(* Logix 5000 project; controller AdvManLab vendor 1 type 14 code 158 rev 28.12; software revision 28.01; part 7 of 13 *)
(* tags used below, declared in another part *)
   R6Z_Current_Part_NO : SINT;
   R6Z_Current_Process_NO : SINT;
   R6Z_Process : BOOL;
   R6Z_Read : BOOL;
   R6Z_Read_Finished : BOOL;
   R6Z_Write_Pass : BOOL;
   ABBLoopVFD : PF525_Faceplate_AOI;
   BobsBits : DINT;
   C21PartInTransit : TIMER;
   C23PartInTransit : TIMER;
   C2HoldBack : PalletStop;
   C2RobotStop : PalletStop;
   C2RobotStopPalletTransit : TIMER;
   C2RobotStopRetractConditions : BOOL;
   C31DiverterHoldBack : PalletStop;
   C31PartInTransit : TIMER;
   Cell_2 : Fanuc_Cell;
   Cloud_R1Z_TagPresent : BOOL;
   Cloud_R1Z_Timer : TIMER;
   Cloud_R2Z_TagPresent : BOOL;
   Cloud_R2Z_Timer : TIMER;
   Cloud_R3Z_TagPresent : BOOL;
   Cloud_R3Z_Timer : TIMER;
   Cloud_R4Z_TagPresent : BOOL;
   Cloud_R4Z_Timer : TIMER;
   Cloud_R5Z_TagPresent : BOOL;
   Cloud_R5Z_Timer : TIMER;
   Cloud_R6Z_TagPresent : BOOL;
   Cloud_R6Z_Timer : TIMER;
   CNC1Bools : DINT;
   CNC2Bools : DINT;
   CNC3Bools : DINT;
   CNC_1_ProgToRun : DINT;
   CNC_2_ProgToRun : DINT;   // G-Code Program Number for CNC to run TO CNC
   CNC_3_Done : BOOL;   // CNC 3 has completed cutting the part
   CNC_3_ProgToRun : DINT;   // G-code program number to be paassed to CNC to run
   CNC_4_Done : BOOL;   // CNC 4 has completed cutting the part
   Comm_Fault_Sts_Timer2 : TIMER;
   Comm_Status : DINT;
   Comm_Status2 : DINT;
   DeBounce3 : TIMER;
   DeBounce4 : TIMER;
   Fault_Code2 : DINT;
   FaultReset : BOOL;
   FltMsg2 : MESSAGE;
   FromCNC1 : CNC_Datablock;   // Data From CNC1
   FromCNC2 : CNC_Datablock;   // Data From CNC2
   FromCNC3 : CNC_Datablock;   // Data From CNC3
   FromCNC4 : CNC_Datablock;   // Data From CNC4
   HMI_Mode : DINT;
   Mode_Auto : BOOL;
   Mode_Semi : BOOL;
   Mode_Start : BOOL;
   ONS : DINT;
   PF525_AlarmName2 : STRING;
   PowerFlexAlarmName2 : STRING;
   PowerFlexAlarmTrigger2 : DINT;
   PPX2 : ALIAS FOR Conv_N053:3:I.0;   // Sensor Pallet Stop RFID2 (Cell 2 Hold Back Stop)
   PPX3 : ALIAS FOR Conv_N053:3:I.1;   // Sensor Pallet Stop RFID3 (Cell 2 Fanuc Robot Stop)
   R2Z_Read_Finished : BOOL;
   R3J_Current_Part_NO : SINT;
   R3J_Current_Process_NO : SINT;
   R3J_Read_Finished : BOOL;
   R3J_Write_Pass : BOOL;
   RelC2HoldBack : TIMER;
   RFIDTP1 : ALIAS FOR RFID_N054:I.Channel[0].TagPresent;   // RFID Tag at Cell 1 Stop
   RFIDTP2 : ALIAS FOR RFID_N054:I.Channel[1].TagPresent;   // RFID Tag at Cell 2 Hold Back Stop
   RFIDTP3 : ALIAS FOR RFID_N055:I.Channel[0].TagPresent;   // RFID Tag at Cell 2 Stop
   RFIDTP4 : ALIAS FOR RFID_N055:I.Channel[1].TagPresent;   // RFID Tag at Cell C23 Hold Back Stop
   RFIDTP5 : ALIAS FOR RFID_N056:I.Channel[0].TagPresent;   // RFID Tag at Cell 3 Stop
   RFIDTP6 : ALIAS FOR RFID_N056:I.Channel[1].TagPresent;
   Robot1_Busy_ZZ : BOOL;
   Robot2_Busy_ZZ : BOOL;
   RunPartOnCNC1 : BOOL;
   RunPartOnCNC2 : BOOL;
   RunpartOnCNC3 : BOOL;
   RunPartOnCNC4 : BOOL;
   ToCNC1 : CNC_Datablock;   // Data To CNC1
   ToCNC2 : CNC_Datablock;   // Data To CNC2
   ToCNC3 : CNC_Datablock;   // Data To CNC3
(* MainProgram, continued *)

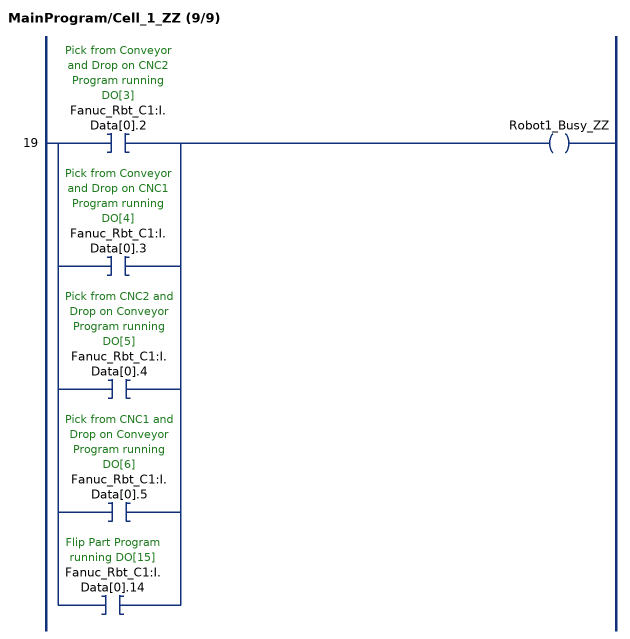
   [picture p119: MainProgram/Cell_1_ZZ rungs 19-19]
   19: [XIC(Fanuc_Rbt_C1:I.Data[0].2) ,XIC(Fanuc_Rbt_C1:I.Data[0].3) ,XIC(Fanuc_Rbt_C1:I.Data[0].4) ,XIC(Fanuc_Rbt_C1:I.Data[0].5) ,XIC(Fanuc_Rbt_C1:I.Data[0].14) ]OTE(Robot1_Busy_ZZ);
END_ROUTINE

ROUTINE Cell_2_ZZ   (* ladder *)
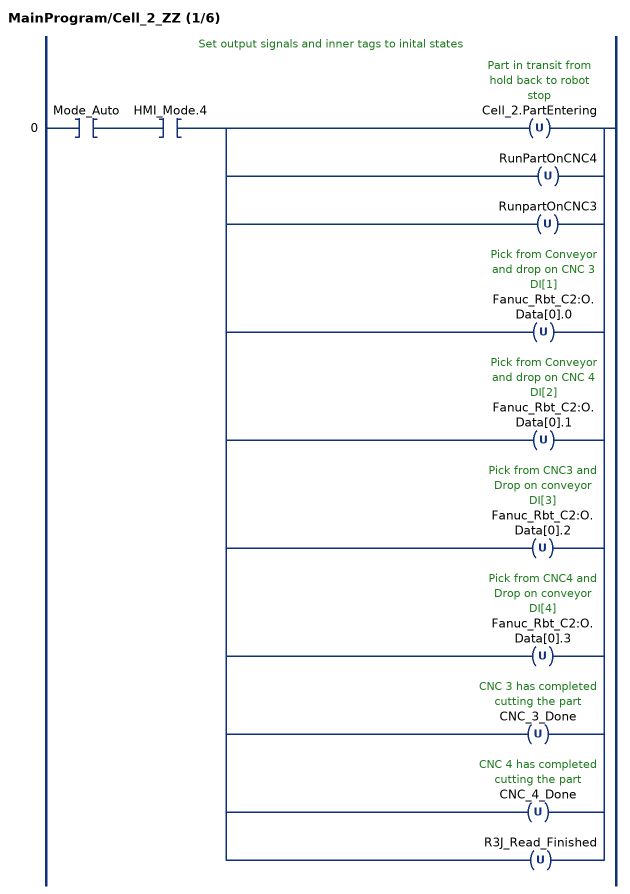
   // Set output signals and inner tags to inital states
   0: XIC(Mode_Auto)XIC(HMI_Mode.4)[OTU(Cell_2.PartEntering) ,OTU(RunPartOnCNC4) ,OTU(RunpartOnCNC3) ,OTU(Fanuc_Rbt_C2:O.Data[0].0) ,OTU(Fanuc_Rbt_C2:O.Data[0].1) ,OTU(Fanuc_Rbt_C2:O.Data[0].2) ,OTU(Fanuc_Rbt_C2:O.Data[0].3) ,OTU(CNC_3_Done) ,OTU(CNC_4_Done) ,OTU(R3J_Read_Finished) ];
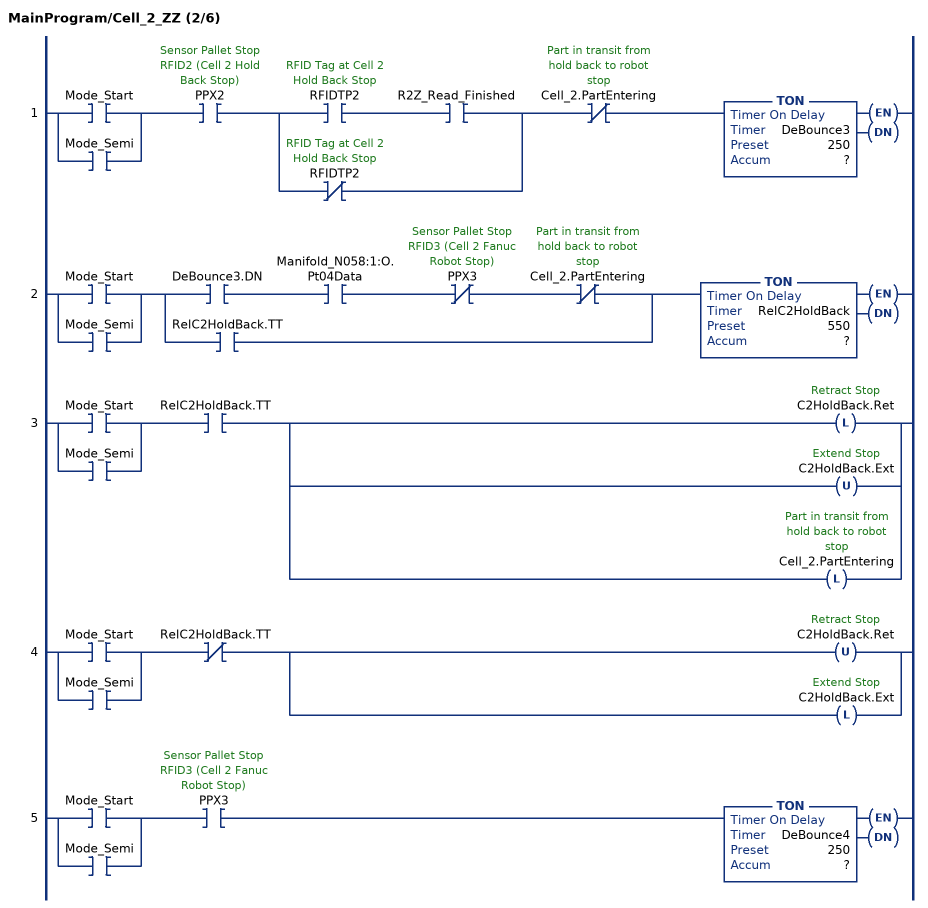
   1: [XIC(Mode_Start) ,XIC(Mode_Semi) ]XIC(PPX2)[XIC(RFIDTP2) XIC(R2Z_Read_Finished) ,XIO(RFIDTP2) ]XIO(Cell_2.PartEntering)TON(DeBounce3,?,?);
   2: [XIC(Mode_Start) ,XIC(Mode_Semi) ][XIC(DeBounce3.DN) XIC(Manifold_N058:1:O.Pt04Data) XIO(PPX3) XIO(Cell_2.PartEntering) ,XIC(RelC2HoldBack.TT) ]TON(RelC2HoldBack,?,?);
   3: [XIC(Mode_Start) ,XIC(Mode_Semi) ]XIC(RelC2HoldBack.TT)[OTL(C2HoldBack.Ret) ,OTU(C2HoldBack.Ext) ,OTL(Cell_2.PartEntering) ];
   4: [XIC(Mode_Start) ,XIC(Mode_Semi) ]XIO(RelC2HoldBack.TT)[OTU(C2HoldBack.Ret) ,OTL(C2HoldBack.Ext) ];
   5: [XIC(Mode_Start) ,XIC(Mode_Semi) ]XIC(PPX3)TON(DeBounce4,?,?);
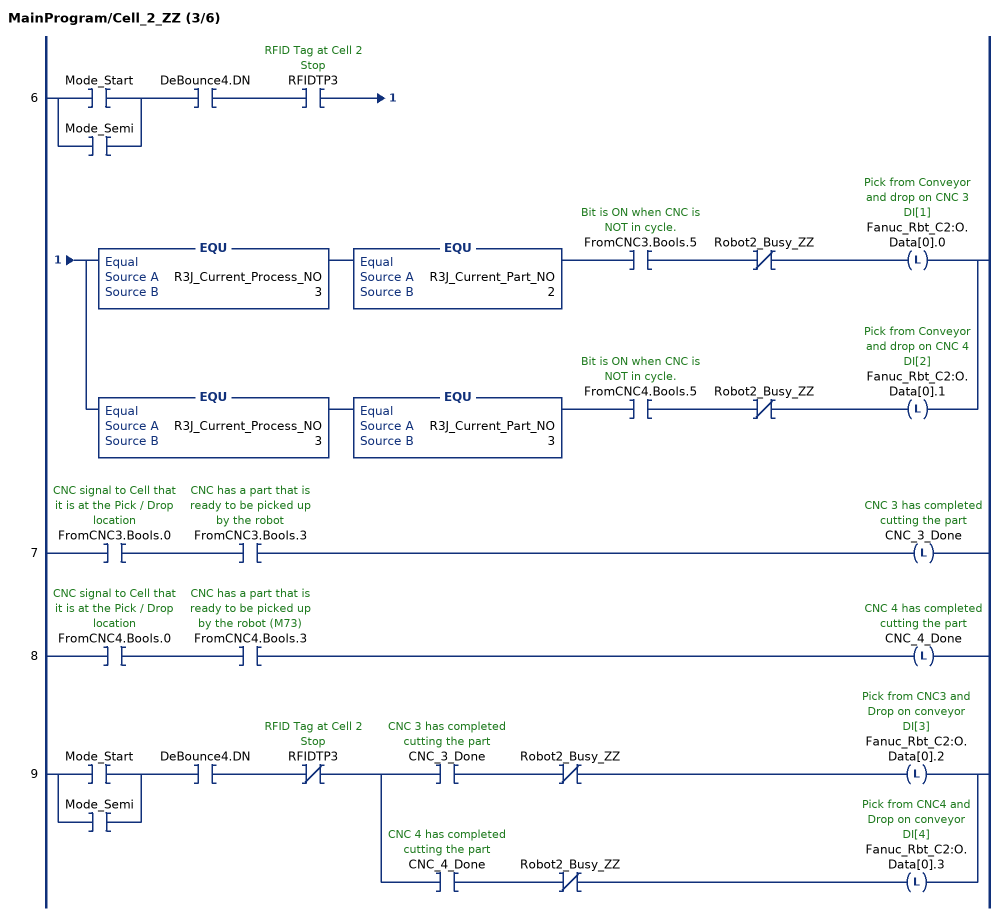
   6: [XIC(Mode_Start) ,XIC(Mode_Semi) ]XIC(DeBounce4.DN)XIC(RFIDTP3)[EQU(R3J_Current_Process_NO,3) EQU(R3J_Current_Part_NO,2) XIC(FromCNC3.Bools.5) XIO(Robot2_Busy_ZZ) OTL(Fanuc_Rbt_C2:O.Data[0].0) ,EQU(R3J_Current_Process_NO,3) EQU(R3J_Current_Part_NO,3) XIC(FromCNC4.Bools.5) XIO(Robot2_Busy_ZZ) OTL(Fanuc_Rbt_C2:O.Data[0].1) ];
   7: XIC(FromCNC3.Bools.0)XIC(FromCNC3.Bools.3)OTL(CNC_3_Done);
   8: XIC(FromCNC4.Bools.0)XIC(FromCNC4.Bools.3)OTL(CNC_4_Done);
   9: [XIC(Mode_Start) ,XIC(Mode_Semi) ]XIC(DeBounce4.DN)XIO(RFIDTP3)[XIC(CNC_3_Done) XIO(Robot2_Busy_ZZ) OTL(Fanuc_Rbt_C2:O.Data[0].2) ,XIC(CNC_4_Done) XIO(Robot2_Busy_ZZ) OTL(Fanuc_Rbt_C2:O.Data[0].3) ];
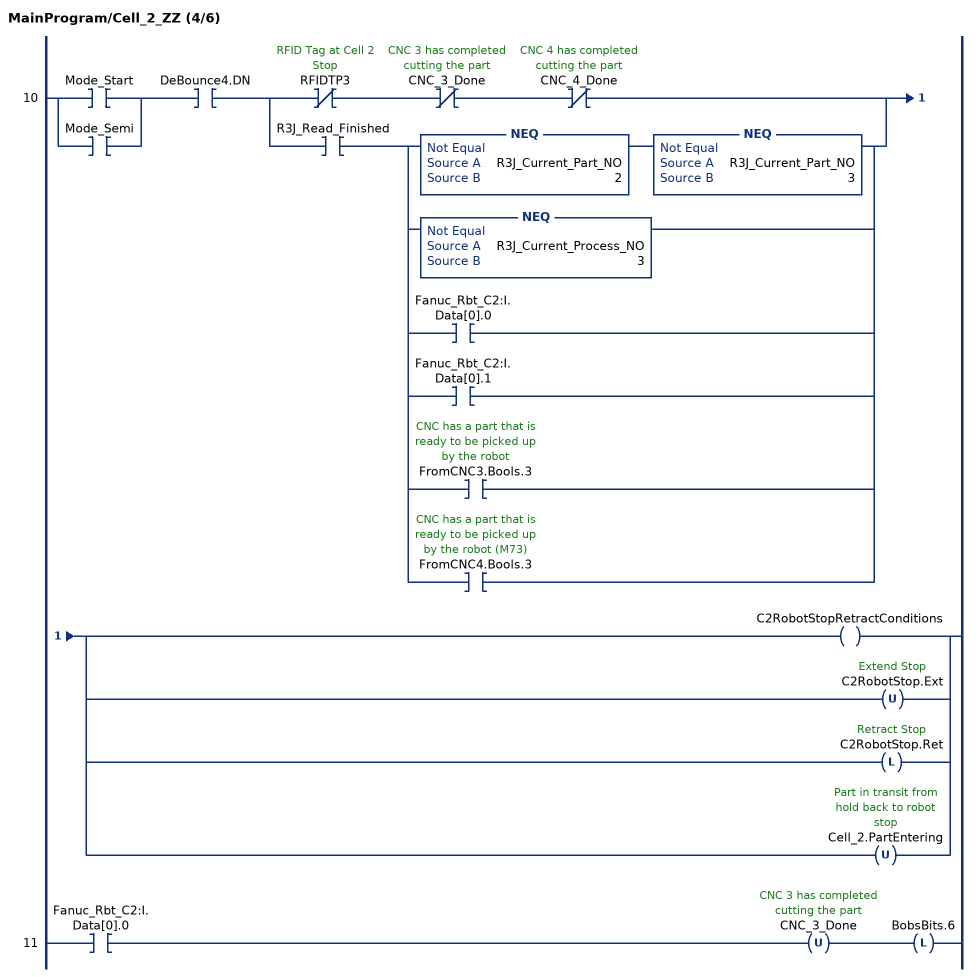
   10: [XIC(Mode_Start) ,XIC(Mode_Semi) ]XIC(DeBounce4.DN)[XIO(RFIDTP3) XIO(CNC_3_Done) XIO(CNC_4_Done) ,XIC(R3J_Read_Finished) [NEQ(R3J_Current_Part_NO,2) NEQ(R3J_Current_Part_NO,3) ,NEQ(R3J_Current_Process_NO,3) ,XIC(Fanuc_Rbt_C2:I.Data[0].0) ,XIC(Fanuc_Rbt_C2:I.Data[0].1) ,[XIC(FromCNC3.Bools.3) ,XIC(FromCNC4.Bools.3) ] ] ][OTE(C2RobotStopRetractConditions) ,OTU(C2RobotStop.Ext) ,OTL(C2RobotStop.Ret) ,OTU(Cell_2.PartEntering) ];
   11: XIC(Fanuc_Rbt_C2:I.Data[0].0)OTU(CNC_3_Done)OTL(BobsBits.6);
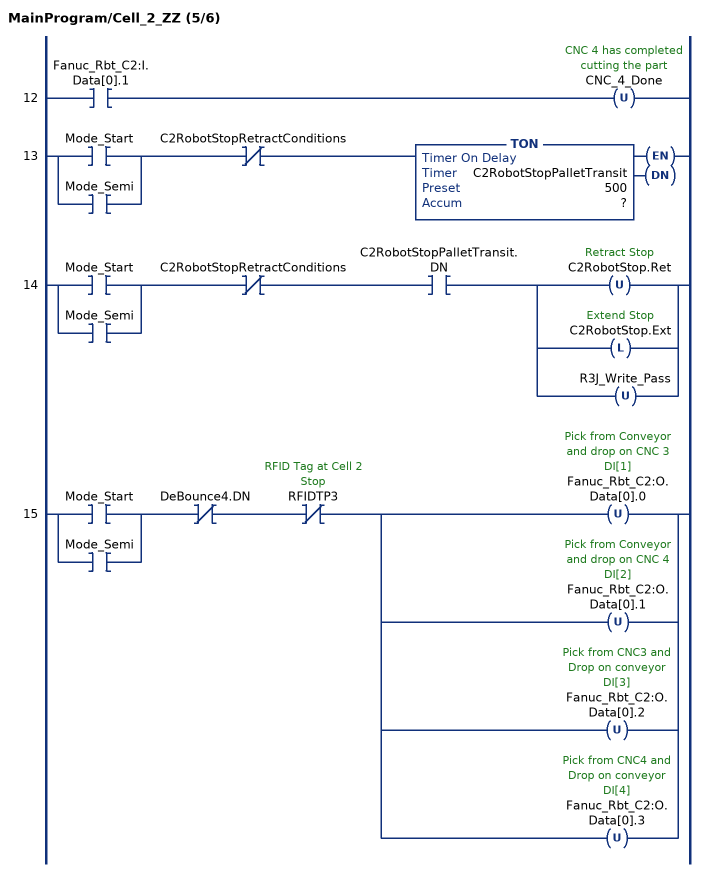
   12: XIC(Fanuc_Rbt_C2:I.Data[0].1)OTU(CNC_4_Done);
   13: [XIC(Mode_Start) ,XIC(Mode_Semi) ]XIO(C2RobotStopRetractConditions)TON(C2RobotStopPalletTransit,?,?);
   14: [XIC(Mode_Start) ,XIC(Mode_Semi) ]XIO(C2RobotStopRetractConditions)XIC(C2RobotStopPalletTransit.DN)[OTU(C2RobotStop.Ret) ,OTL(C2RobotStop.Ext) ,OTU(R3J_Write_Pass) ];
   15: [XIC(Mode_Start) ,XIC(Mode_Semi) ]XIO(DeBounce4.DN)XIO(RFIDTP3)[OTU(Fanuc_Rbt_C2:O.Data[0].0) ,OTU(Fanuc_Rbt_C2:O.Data[0].1) ,OTU(Fanuc_Rbt_C2:O.Data[0].2) ,OTU(Fanuc_Rbt_C2:O.Data[0].3) ];
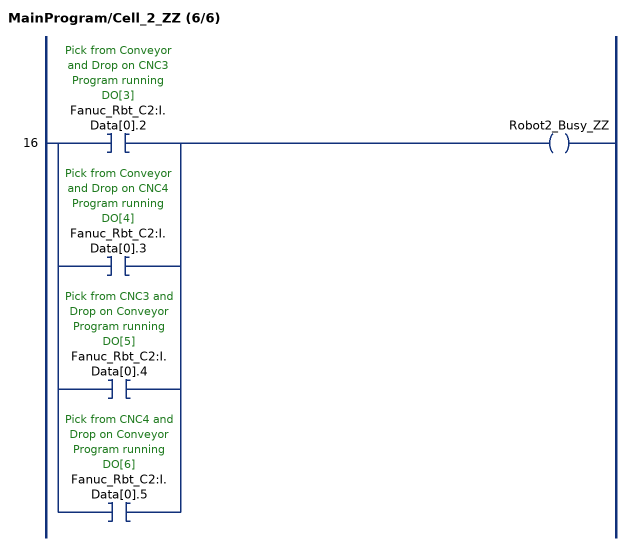
   16: [XIC(Fanuc_Rbt_C2:I.Data[0].2) ,XIC(Fanuc_Rbt_C2:I.Data[0].3) ,XIC(Fanuc_Rbt_C2:I.Data[0].4) ,XIC(Fanuc_Rbt_C2:I.Data[0].5) ]OTE(Robot2_Busy_ZZ);
END_ROUTINE

ROUTINE Cell_3_VFD   (* ladder *)
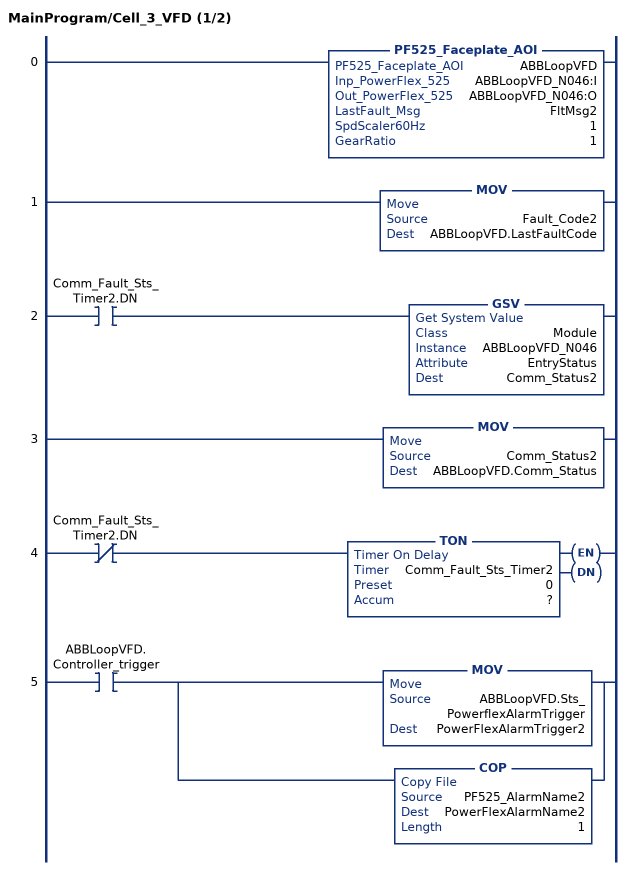
   0: PF525_Faceplate_AOI(ABBLoopVFD,ABBLoopVFD_N046:I,ABBLoopVFD_N046:O,FltMsg2,1,1);
   1: MOV(Fault_Code2,ABBLoopVFD.LastFaultCode);
   2: XIC(Comm_Fault_Sts_Timer2.DN)GSV(Module,ABBLoopVFD_N046,EntryStatus,Comm_Status2);
   3: MOV(Comm_Status2,ABBLoopVFD.Comm_Status);
   4: XIO(Comm_Fault_Sts_Timer2.DN)TON(Comm_Fault_Sts_Timer2,?,?);
   5: XIC(ABBLoopVFD.Controller_trigger)[MOV(ABBLoopVFD.Sts_PowerflexAlarmTrigger,PowerFlexAlarmTrigger2) ,COP(PF525_AlarmName2,PowerFlexAlarmName2,1) ];
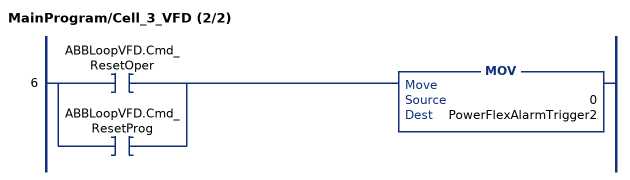
   6: [XIC(ABBLoopVFD.Cmd_ResetOper) ,XIC(ABBLoopVFD.Cmd_ResetProg) ]MOV(0,PowerFlexAlarmTrigger2);
END_ROUTINE

ROUTINE Cell_3_ZZ   (* ladder *)
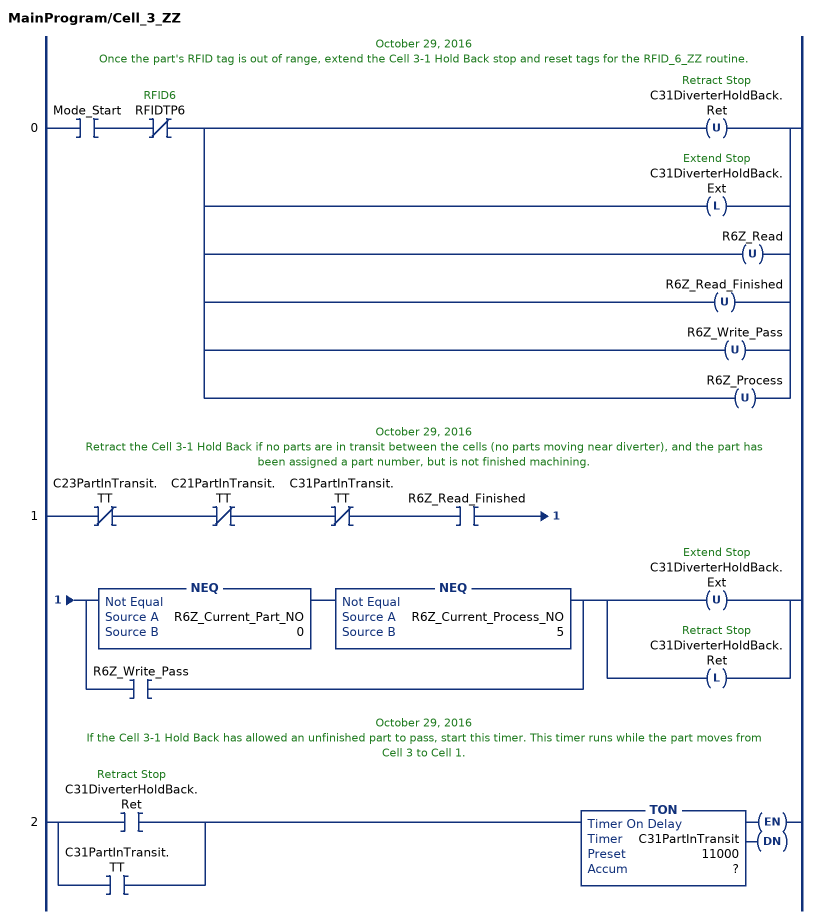
   // October 29, 2016
   // Once the part's RFID tag is out of range, extend the Cell 3-1 Hold Back stop and reset tags for the RFID_6_ZZ routine.
   0: XIC(Mode_Start)XIO(RFIDTP6)[OTU(C31DiverterHoldBack.Ret) ,OTL(C31DiverterHoldBack.Ext) ,OTU(R6Z_Read) ,OTU(R6Z_Read_Finished) ,OTU(R6Z_Write_Pass) ,OTU(R6Z_Process) ];
   // October 29, 2016
   // Retract the Cell 3-1 Hold Back if no parts are in transit between the cells (no parts moving near diverter), and the part has been assigned a part number, but is not finished machining.
   1: XIO(C23PartInTransit.TT)XIO(C21PartInTransit.TT)XIO(C31PartInTransit.TT)XIC(R6Z_Read_Finished)[NEQ(R6Z_Current_Part_NO,0) NEQ(R6Z_Current_Process_NO,5) ,XIC(R6Z_Write_Pass) ][OTU(C31DiverterHoldBack.Ext) ,OTL(C31DiverterHoldBack.Ret) ];
   // October 29, 2016
   // If the Cell 3-1 Hold Back has allowed an unfinished part to pass, start this timer. This timer runs while the part moves from Cell 3 to Cell 1.
   2: [XIC(C31DiverterHoldBack.Ret) ,XIC(C31PartInTransit.TT) ]TON(C31PartInTransit,?,?);
END_ROUTINE

ROUTINE Cloud_Team_ZZ   (* ladder *)
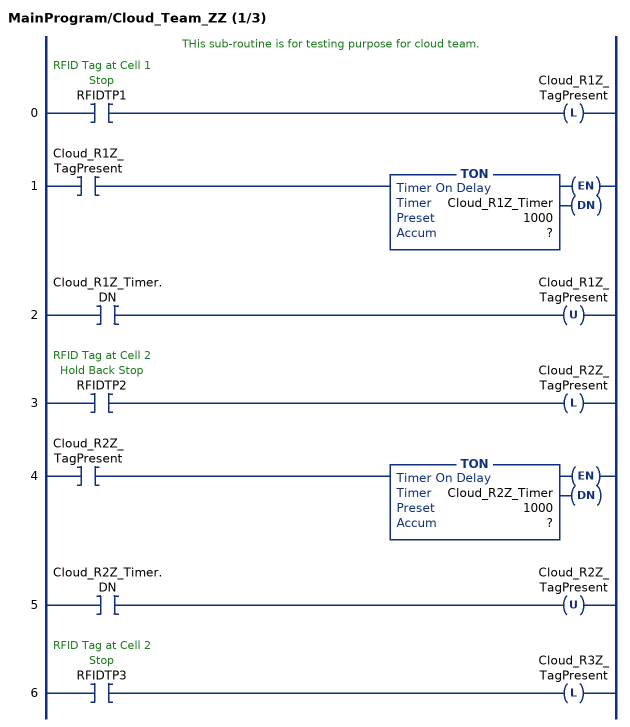
   // THis sub-routine is for testing purpose for cloud team.
   0: XIC(RFIDTP1)OTL(Cloud_R1Z_TagPresent);
   1: XIC(Cloud_R1Z_TagPresent)TON(Cloud_R1Z_Timer,?,?);
   2: XIC(Cloud_R1Z_Timer.DN)OTU(Cloud_R1Z_TagPresent);
   3: XIC(RFIDTP2)OTL(Cloud_R2Z_TagPresent);
   4: XIC(Cloud_R2Z_TagPresent)TON(Cloud_R2Z_Timer,?,?);
   5: XIC(Cloud_R2Z_Timer.DN)OTU(Cloud_R2Z_TagPresent);
   6: XIC(RFIDTP3)OTL(Cloud_R3Z_TagPresent);
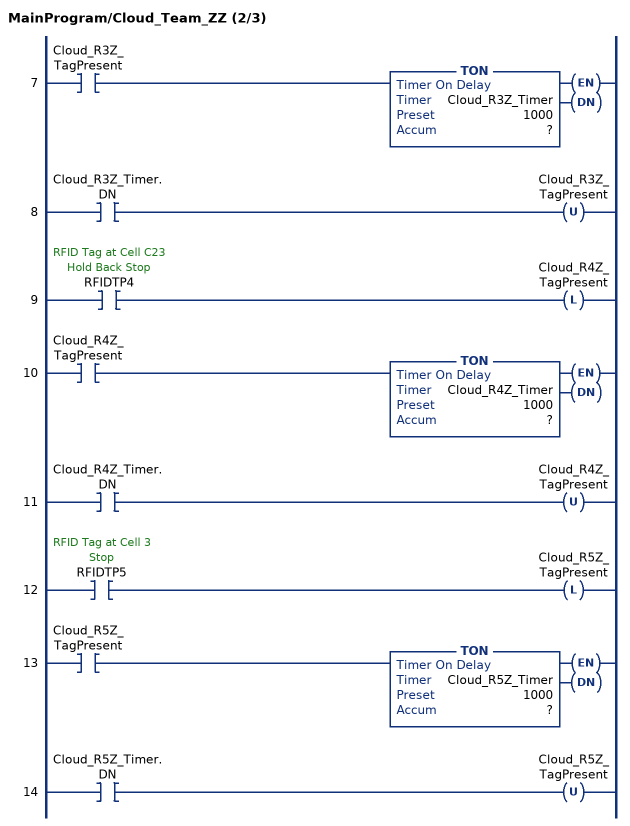
   7: XIC(Cloud_R3Z_TagPresent)TON(Cloud_R3Z_Timer,?,?);
   8: XIC(Cloud_R3Z_Timer.DN)OTU(Cloud_R3Z_TagPresent);
   9: XIC(RFIDTP4)OTL(Cloud_R4Z_TagPresent);
   10: XIC(Cloud_R4Z_TagPresent)TON(Cloud_R4Z_Timer,?,?);
   11: XIC(Cloud_R4Z_Timer.DN)OTU(Cloud_R4Z_TagPresent);
   12: XIC(RFIDTP5)OTL(Cloud_R5Z_TagPresent);
   13: XIC(Cloud_R5Z_TagPresent)TON(Cloud_R5Z_Timer,?,?);
   14: XIC(Cloud_R5Z_Timer.DN)OTU(Cloud_R5Z_TagPresent);
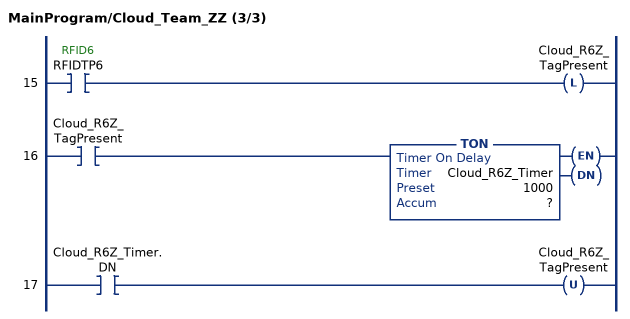
   15: XIC(RFIDTP6)OTL(Cloud_R6Z_TagPresent);
   16: XIC(Cloud_R6Z_TagPresent)TON(Cloud_R6Z_Timer,?,?);
   17: XIC(Cloud_R6Z_Timer.DN)OTU(Cloud_R6Z_TagPresent);
END_ROUTINE

ROUTINE CNC1   (* ladder *)
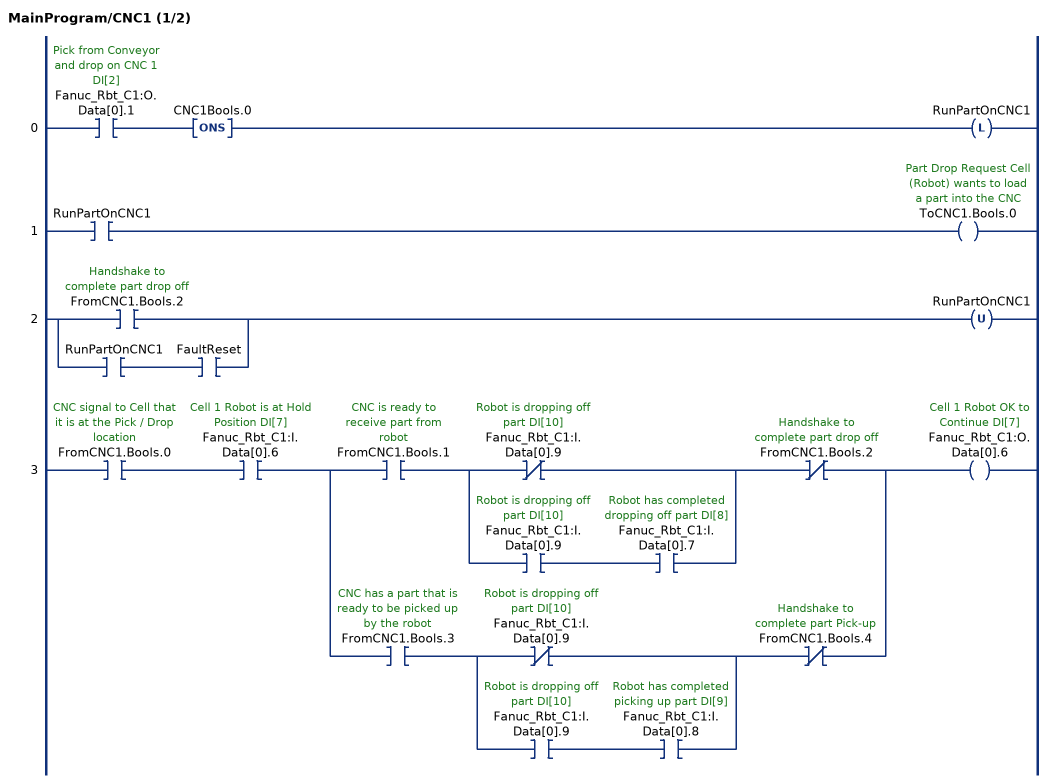
   0: XIC(Fanuc_Rbt_C1:O.Data[0].1)ONS(CNC1Bools.0)OTL(RunPartOnCNC1);
   1: XIC(RunPartOnCNC1)OTE(ToCNC1.Bools.0);
   2: [XIC(FromCNC1.Bools.2) ,XIC(RunPartOnCNC1) XIC(FaultReset) ]OTU(RunPartOnCNC1);
   3: XIC(FromCNC1.Bools.0)XIC(Fanuc_Rbt_C1:I.Data[0].6)[XIC(FromCNC1.Bools.1) [XIO(Fanuc_Rbt_C1:I.Data[0].9) ,XIC(Fanuc_Rbt_C1:I.Data[0].9) XIC(Fanuc_Rbt_C1:I.Data[0].7) ] XIO(FromCNC1.Bools.2) ,XIC(FromCNC1.Bools.3) [XIO(Fanuc_Rbt_C1:I.Data[0].9) ,XIC(Fanuc_Rbt_C1:I.Data[0].9) XIC(Fanuc_Rbt_C1:I.Data[0].8) ] XIO(FromCNC1.Bools.4) ]OTE(Fanuc_Rbt_C1:O.Data[0].6);
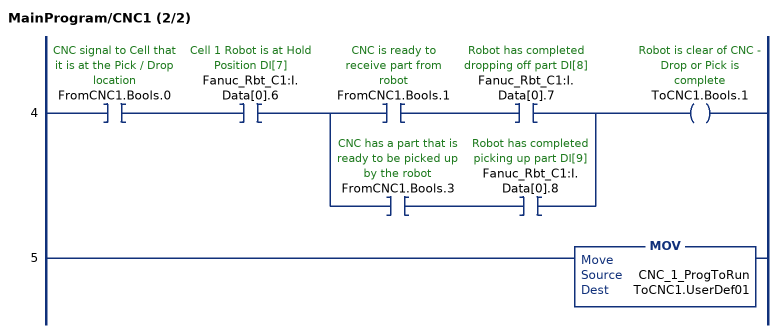
   4: XIC(FromCNC1.Bools.0)XIC(Fanuc_Rbt_C1:I.Data[0].6)[XIC(FromCNC1.Bools.1) XIC(Fanuc_Rbt_C1:I.Data[0].7) ,XIC(FromCNC1.Bools.3) XIC(Fanuc_Rbt_C1:I.Data[0].8) ]OTE(ToCNC1.Bools.1);
   5: MOV(CNC_1_ProgToRun,ToCNC1.UserDef01);
END_ROUTINE

ROUTINE CNC2   (* ladder *)
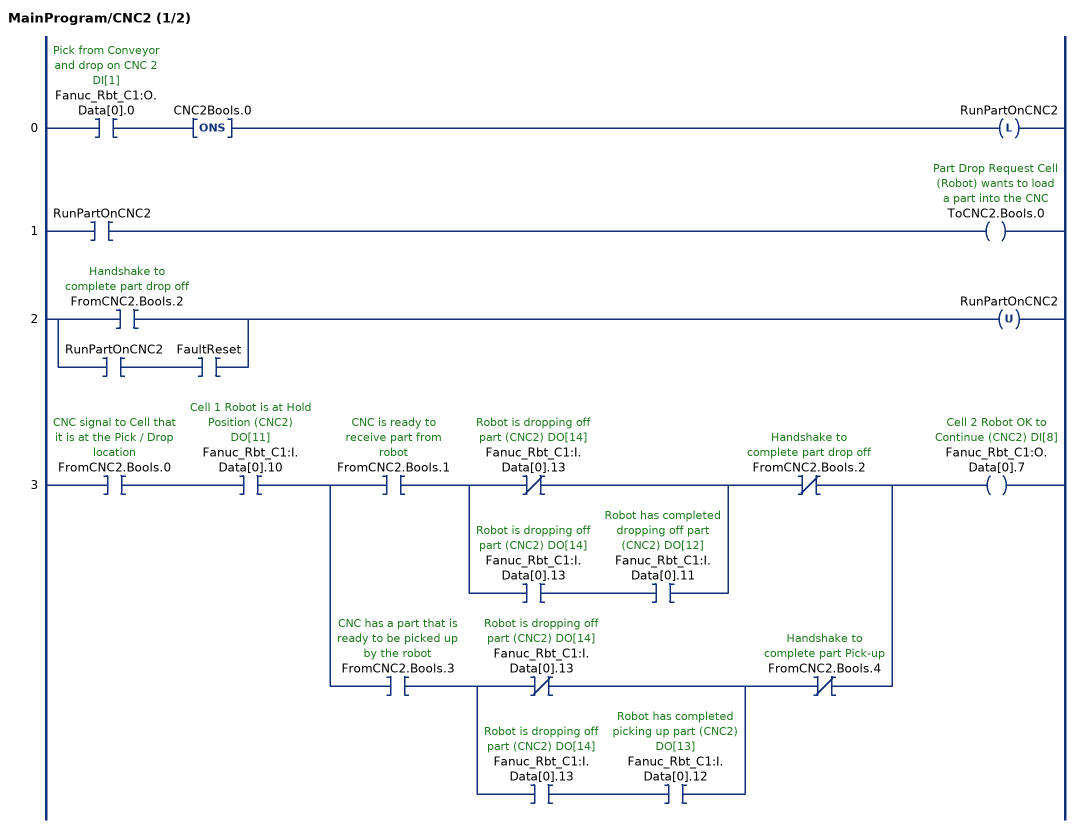
   0: XIC(Fanuc_Rbt_C1:O.Data[0].0)ONS(CNC2Bools.0)OTL(RunPartOnCNC2);
   1: XIC(RunPartOnCNC2)OTE(ToCNC2.Bools.0);
   2: [XIC(FromCNC2.Bools.2) ,XIC(RunPartOnCNC2) XIC(FaultReset) ]OTU(RunPartOnCNC2);
   3: XIC(FromCNC2.Bools.0)XIC(Fanuc_Rbt_C1:I.Data[0].10)[XIC(FromCNC2.Bools.1) [XIO(Fanuc_Rbt_C1:I.Data[0].13) ,XIC(Fanuc_Rbt_C1:I.Data[0].13) XIC(Fanuc_Rbt_C1:I.Data[0].11) ] XIO(FromCNC2.Bools.2) ,XIC(FromCNC2.Bools.3) [XIO(Fanuc_Rbt_C1:I.Data[0].13) ,XIC(Fanuc_Rbt_C1:I.Data[0].13) XIC(Fanuc_Rbt_C1:I.Data[0].12) ] XIO(FromCNC2.Bools.4) ]OTE(Fanuc_Rbt_C1:O.Data[0].7);
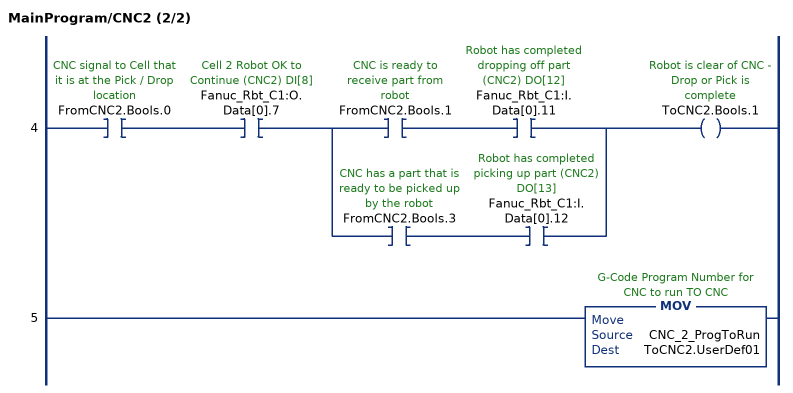
   4: XIC(FromCNC2.Bools.0)XIC(Fanuc_Rbt_C1:O.Data[0].7)[XIC(FromCNC2.Bools.1) XIC(Fanuc_Rbt_C1:I.Data[0].11) ,XIC(FromCNC2.Bools.3) XIC(Fanuc_Rbt_C1:I.Data[0].12) ]OTE(ToCNC2.Bools.1);
   5: MOV(CNC_2_ProgToRun,ToCNC2.UserDef01);
END_ROUTINE

ROUTINE CNC3   (* ladder *)
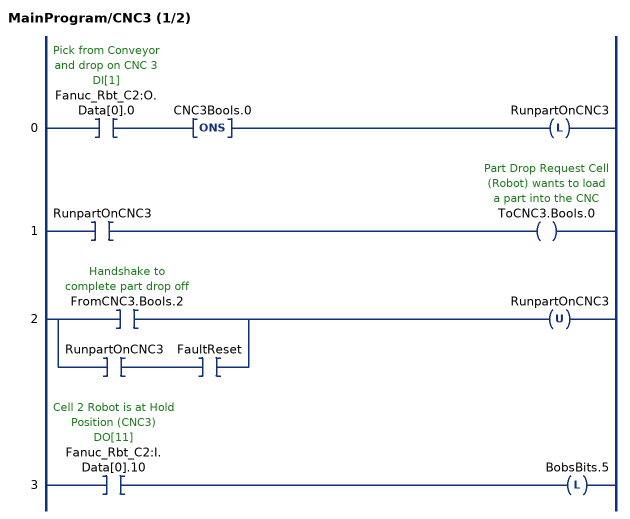
   0: XIC(Fanuc_Rbt_C2:O.Data[0].0)ONS(CNC3Bools.0)OTL(RunpartOnCNC3);
   1: XIC(RunpartOnCNC3)OTE(ToCNC3.Bools.0);
   2: [XIC(FromCNC3.Bools.2) ,XIC(RunpartOnCNC3) XIC(FaultReset) ]OTU(RunpartOnCNC3);
   3: XIC(Fanuc_Rbt_C2:I.Data[0].10)OTL(BobsBits.5);
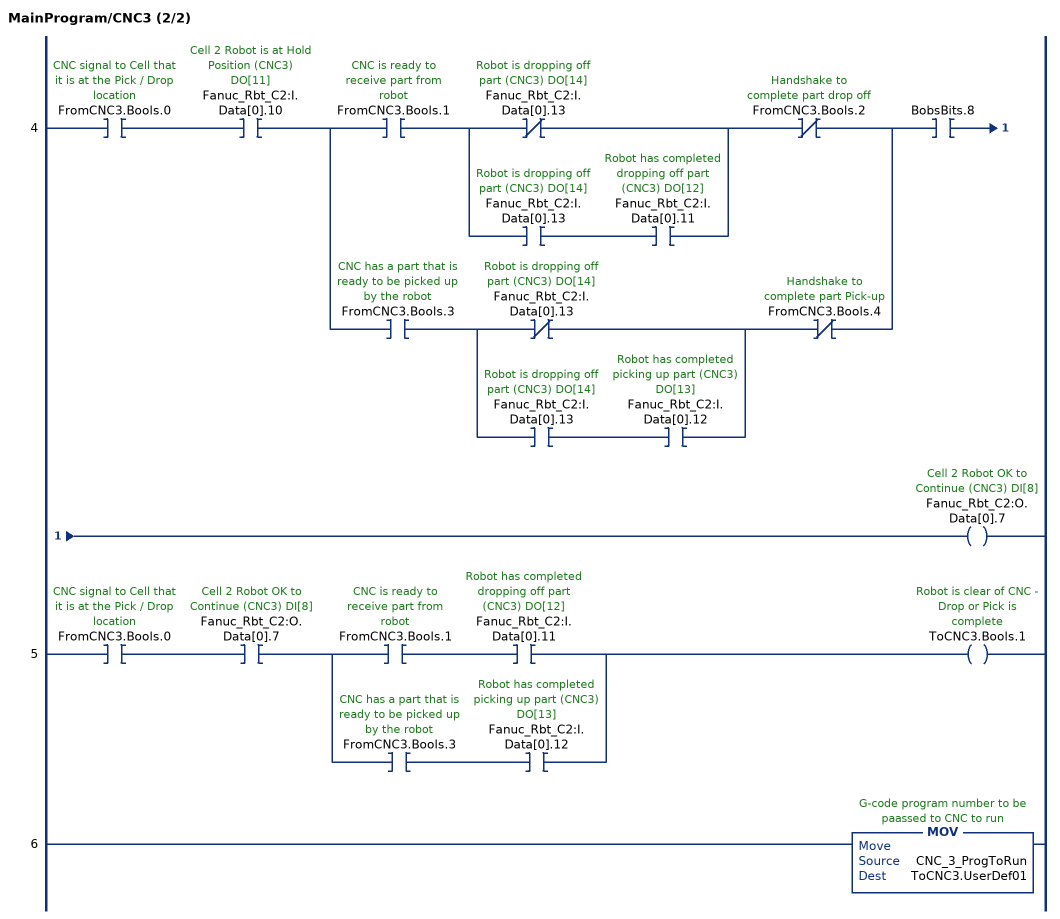
   4: XIC(FromCNC3.Bools.0)XIC(Fanuc_Rbt_C2:I.Data[0].10)[XIC(FromCNC3.Bools.1) [XIO(Fanuc_Rbt_C2:I.Data[0].13) ,XIC(Fanuc_Rbt_C2:I.Data[0].13) XIC(Fanuc_Rbt_C2:I.Data[0].11) ] XIO(FromCNC3.Bools.2) ,XIC(FromCNC3.Bools.3) [XIO(Fanuc_Rbt_C2:I.Data[0].13) ,XIC(Fanuc_Rbt_C2:I.Data[0].13) XIC(Fanuc_Rbt_C2:I.Data[0].12) ] XIO(FromCNC3.Bools.4) ]XIC(BobsBits.8)OTE(Fanuc_Rbt_C2:O.Data[0].7);
   5: XIC(FromCNC3.Bools.0)XIC(Fanuc_Rbt_C2:O.Data[0].7)[XIC(FromCNC3.Bools.1) XIC(Fanuc_Rbt_C2:I.Data[0].11) ,XIC(FromCNC3.Bools.3) XIC(Fanuc_Rbt_C2:I.Data[0].12) ]OTE(ToCNC3.Bools.1);
   6: MOV(CNC_3_ProgToRun,ToCNC3.UserDef01);
END_ROUTINE
